{attribute addProperty BoxType "EL9221-4030-0018"}
{attribute addProperty Id "OCP_InputsAT %I*OCP_Inputs_FE08AF3C3240OCP_OutputsAT %Q*OCP_Outputs_F330A9161620WcStateAT %I*WcState_98A4DF7520.250InfoDataAT %I*InfoData_BC63D37F80100"}
{attribute addProperty CRC "2904856186"}
{attribute addProperty SizeInBites "130"}
{attribute addProperty SizeInBytes "16.25"}
TYPE EL9221_E4BC0073 :
STRUCT
	{attribute addProperty Name "OCP_Inputs"}
	OCP_Inputs : OCP_Inputs_FE08AF3C;
	{attribute addProperty Name "OCP_Outputs"}
	OCP_Outputs : OCP_Outputs_F330A916;
	{attribute addProperty Name "WcState"}
	WcState : WcState_98A4DF75;
	{attribute addProperty Name "InfoData"}
	InfoData : InfoData_BC63D37F;
END_STRUCT
END_TYPE

(* stored: Version 1.2.0.0, ProductVersion 3.1.4024.9
   DUT EL9221_E4BC0073: Id {407cad3b-3384-4e0d-820b-48ad39d13e15} *)
